{attribute 'qualified_only'}
VAR_GLOBAL
	sNetId: T_AmsNetId := '5.30.23.91.1.1';
	nPort: T_AmsPort := 851;	
END_VAR

(* stored: Version 1.1.0.1, ProductVersion 3.1.4024.11
   GVL SUPVams: Id {589d3e13-63d8-4473-8161-8704225dc42b} *)
